FUNCTION_BLOCK FB_SPINDLE
VAR_INPUT
END_VAR
VAR_OUTPUT
END_VAR
VAR
	pbToolChange AT %I*: BOOL;
	changeToolEnable: BOOL;
	cylinderToolRelease1 AT %Q* : BOOL;
	cylinderToolRelease2 AT %Q* : BOOL;
	
	toolChangeTimer : TON;
END_VAR

Tool_Change();

METHOD Tool_Change
VAR_INPUT
END_VAR
IF changeToolEnable THEN
	toolChangeTimer(IN:= pbToolChange, PT:=T#2S);
	
	IF pbToolChange THEN
		IF toolChangeTimer.Q THEN
			cylinderToolRelease1 := TRUE;
			cylinderToolRelease2 := TRUE;
		END_IF
	ELSE
		cylinderToolRelease1 := FALSE;
		cylinderToolRelease2 := FALSE;
	END_IF
END_IF
END_METHOD

END_FUNCTION_BLOCK

(* stored: Version 1.1.0.1, ProductVersion 3.1.4024.12
   POU FB_SPINDLE: Id {3dc147eb-3dde-4052-8db8-ee0200a73c1f}, SpecialFunc None
   Method Tool_Change: Id {caf02692-220f-45ea-9a62-11b6af7ca524} *)
